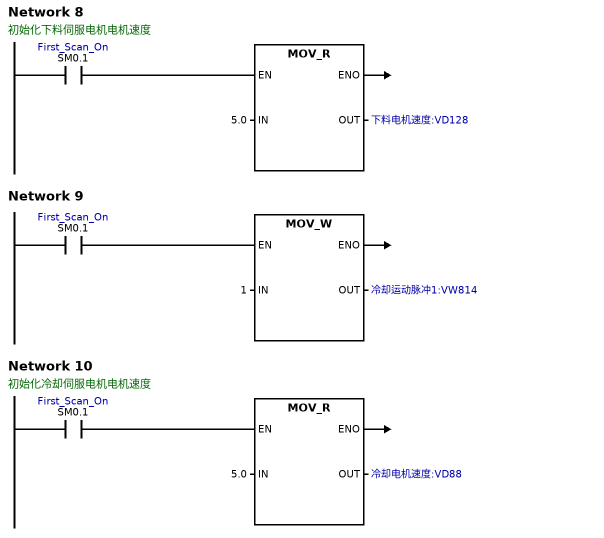
[picture p24: SBR20 networks 8-10]
Network 8
// 初始化下料伺服电机电机速度
LD     First_Scan_On:SM0.1
MOVR   5.0, 下料电机速度:VD128
Network 9
LD     First_Scan_On:SM0.1
MOVW   1, 冷却运动脉冲1:VW814
Network 10
// 初始化冷却伺服电机电机速度
LD     First_Scan_On:SM0.1
MOVR   5.0, 冷却电机速度:VD88
END_SUBROUTINE_BLOCK

SUBROUTINE_BLOCK 故障报警:SBR21
TITLE=子程序注释
BEGIN
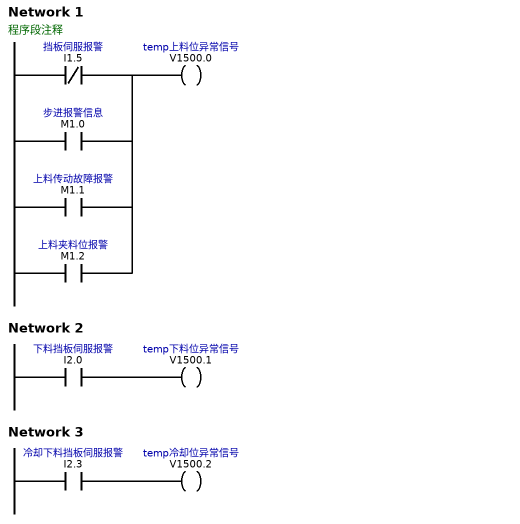
Network 1
// 程序段注释
// (network saved uncompiled; LAD cells follow)
// row 0: c0 -|/|- 挡板伺服报警:I1.5 v  c1 -( ) temp上料位异常信号:V1500.0
// row 1: c0 -| |- 步进报警信息:M1.0 ^v
// row 2: c0 -| |- 上料传动故障报警:M1.1 ^v
// row 3: c0 -| |- 上料夹料位报警:M1.2 ^
Network 2
LD     下料挡板伺服报警:I2.0
=      temp下料位异常信号:V1500.1
Network 3
LD     冷却下料挡板伺服报警:I2.3
=      temp冷却位异常信号:V1500.2
END_SUBROUTINE_BLOCK
